TYPE (* ISO Part 5 name field structure according to IFM conventions *)
  (* Version 1.0, 2025-09-04, Coding-Assistent *)
  PACKAGE isobus;
  NAMEFIELD_T : STRUCT
    bSelfConf : BOOL := TRUE; (* Self-configurable-address ECU? *)
    bIndGroup : BYTE := 16#FF; (* NAMES associated with industries (0..7) *)
    bDevClassInst : BYTE := 16#FF; (* Identifier if a device class more than 1 times in net (0..15) *)
    bDevClass : BYTE := 16#FF; (* ISO Defined (0..127) *)
    bReserved : BOOL := TRUE; (* Reserved (not used) *)
    bFunction : BYTE := 16#FF; (* ISO defined, -> SA (0..255) *)
    bFunctionInst : BYTE := 16#FF; (* Subgroup of function (0..31) *)
    bEcuInstance : BYTE := 16#FF; (* Which ECU associated with a given function (0..7) *)
    wManufCode : WORD := 16#FFFF; (* ISO defined (0..2047) *)
    dwIdentNumb : DWORD := 16#FFFFFFFF; (* Used when the NAME is not unique in same network (0..2047) *)
  END_STRUCT;
END_TYPE
